PROGRAM POU_Interlock
VAR
END_VAR


//Interlock 

//

END_PROGRAM

(* stored: Version 1.1.0.1, ProductVersion 3.1.4022.18
   POU POU_Interlock: Id {a30357a6-8d74-4b6d-bda7-5c5ec5f69b13}, SpecialFunc None *)
